// Mitsubishi GX Works2 project: Test   PLC: FX3G

// global labels: Global1
VAR_GLOBAL
  xStart AT M0 : BOOL;
  xAlarm AT M1 : BOOL;
  xAlarmCritical AT M2 : BOOL;
  xWarning AT M3 : BOOL;
  xInit AT M4 : BOOL;
  aI_TempOut AT D500 : INT;
  dI_PowerOn AT X001 : BOOL;
  dO_SupplyStart AT Y001 : BOOL;
END_VAR

// task Task_01 (event TRUE, interval 0, priority 31): POU_01
// user libraries (not included): AlarmMange, Easings, Utils

PROGRAM POU_01
;
END_PROGRAM

PROGRAM Init
VAR
  fbAmInit : AM_INIT;
  fbAmSet : AM_SET;
  fbAmIs : AM_HAS_ALARMS;
  fbAmBlockIs : AM_IS_BLOCK;
  fbAmReset : AM_RST;
END_VAR
IF NOT xInit THEN
	fbAmInit(iNum:= 0 ,iSeverity:= 2 ,iProcess:= 1 ,xLatch:= FALSE ,xBuzzer:= TRUE , xLock:= TRUE );
	fbAmInit(iNum:= 1 ,iSeverity:= 3 ,iProcess:= 2 ,xLatch:= TRUE ,xBuzzer:= TRUE , xLock:= TRUE );
	xInit := TRUE;	
END_IF;

IF NOT (D8031 = 32760) THEN
	aI_TempOut := SCALE( D8031 , 803 , 1740 , -500 , 1950 );
ELSE
	aI_TempOut := -50;
END_IF;
	
fbAmSet(iNum:= 0 ,xState:= (D8031 = 32760) );
fbAmSet(iNum:= 1 ,xState:= (X000 = 1) );
fbAmIs(iProcessNum:= 0 ,iSeverity:= 2 ,Q:= xAlarm );
fbAmIs(iProcessNum:= 1 ,iSeverity:= 3 ,Q:= xAlarmCritical );
END_PROGRAM
